// TIA Portal V19 export
FUNCTION "HmiButtonColor" : Int   // FC18, LAD
TITLE = CHANGE APPAREANCE IN HMI BUTTONS
// stored: SetENOAutomatically false
   VAR_INPUT
      Permit : Bool;
      InProgress : Bool;
      Done : Bool;
      Error : Bool;
   END_VAR
   VAR CONSTANT
      COLOR_DISABLE : Int := 0;
      COLOR_ENABLE : Int := 1;
      COLOR_IN_PROGRESS : Int := 2;
      COLOR_DONE : Int := 3;
      COLOR_ERROR : Int := 4;
   END_VAR
BEGIN

REGION Network 1: Main
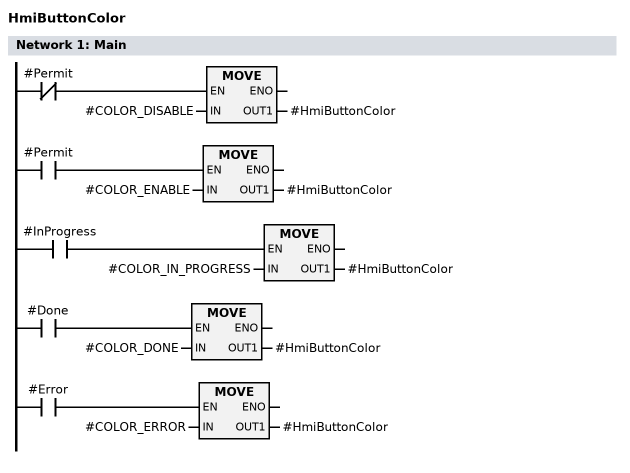
   RUNG wire#powerrail
      I_Contact( #Permit )
      Move(in := #COLOR_DISABLE, out1 => #HmiButtonColor)
   END_RUNG
   RUNG wire#powerrail
      Contact( #Permit )
      Move(in := #COLOR_ENABLE, out1 => #HmiButtonColor)
   END_RUNG
   RUNG wire#powerrail
      Contact( #InProgress )
      Move(in := #COLOR_IN_PROGRESS, out1 => #HmiButtonColor)
   END_RUNG
   RUNG wire#powerrail
      Contact( #Done )
      Move(in := #COLOR_DONE, out1 => #HmiButtonColor)
   END_RUNG
   RUNG wire#powerrail
      Contact( #Error )
      Move(in := #COLOR_ERROR, out1 => #HmiButtonColor)
   END_RUNG
   // the same network as SCL:
   IF NOT #Permit THEN #HmiButtonColor := #COLOR_DISABLE; END_IF;
   IF #Permit THEN #HmiButtonColor := #COLOR_ENABLE; END_IF;
   IF #InProgress THEN #HmiButtonColor := #COLOR_IN_PROGRESS; END_IF;
   IF #Done THEN #HmiButtonColor := #COLOR_DONE; END_IF;
   IF #Error THEN #HmiButtonColor := #COLOR_ERROR; END_IF;
END_REGION
END_FUNCTION
